// TwinCAT 3 PLC project VB_ADS_Sample
// ProgramVersion: 3.1.4026.24
// libraries:
//   Tc2_Standard, * (Beckhoff Automation GmbH)
//   Tc2_System, * (Beckhoff Automation GmbH)
//   Tc3_Module, * (Beckhoff Automation GmbH)
//   VisuSymbols,3.5.10.0,System
// project tree:
//   / GlobalTextList.TcGTLO, PlcTask.TcTTO, Visualization Manager.TcVMO (not stored)
//   POUs/ MAIN.TcPOU
//   VISUs/ Visualization.TcVIS
// real-time tasks:
//   TASK PlcTask: cycle T#10ms, priority 20, ADS port 350

CONFIGURATION VB_ADS_Sample
    RESOURCE PLC ON TwinCAT3
        TASK PlcTask(INTERVAL := T#10ms, PRIORITY := 20);
        PROGRAM MAIN WITH PlcTask : MAIN;
    END_RESOURCE
END_CONFIGURATION

// ---- POUs/MAIN.TcPOU
PROGRAM MAIN
VAR
	test_input AT%I* : ARRAY [0..1] OF BOOL;
	test_output AT%Q* : ARRAY [0..1] OF BOOL;
	test_value : DINT;
	test_string: STRING(255);
END_VAR


IF test_value = 16#7FFFFFFF THEN
	test_value := 0;
END_IF

test_value := test_value + 1;

END_PROGRAM

// ---- GlobalTextList.TcGTLO
TEXTLIST GlobalTextList
  25 = '%0s'
  345 = '%S'
END_TEXTLIST

// ---- VISUs/Visualization.TcVIS
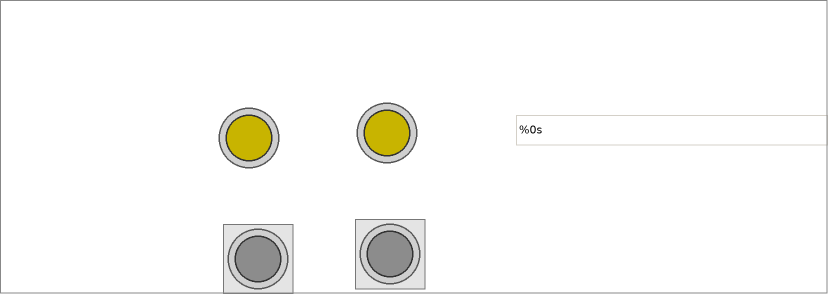
VISUALIZATION Visualization  // 828x294
    Lamp1 (214,103 70x70), variable: MAIN.test_output[0], style: Lamp-Lamp1-Yellow
    PushSwitch (223,224 70x70), variable: MAIN.test_input[0], behaviour: TAP, style: Switch-PushSwitch-Gray
    Lamp1 (352,98 70x70), variable: MAIN.test_output[1], style: Lamp-Lamp1-Yellow
    PushSwitch (355,219 70x70), variable: MAIN.test_input[1], behaviour: TOGGLE, style: Switch-PushSwitch-Gray
    Textfield (516,115 312x30), "%0s", text variable: MAIN.test_string
        OnMouseClick: write the text variable via Edit
END_VISUALIZATION
